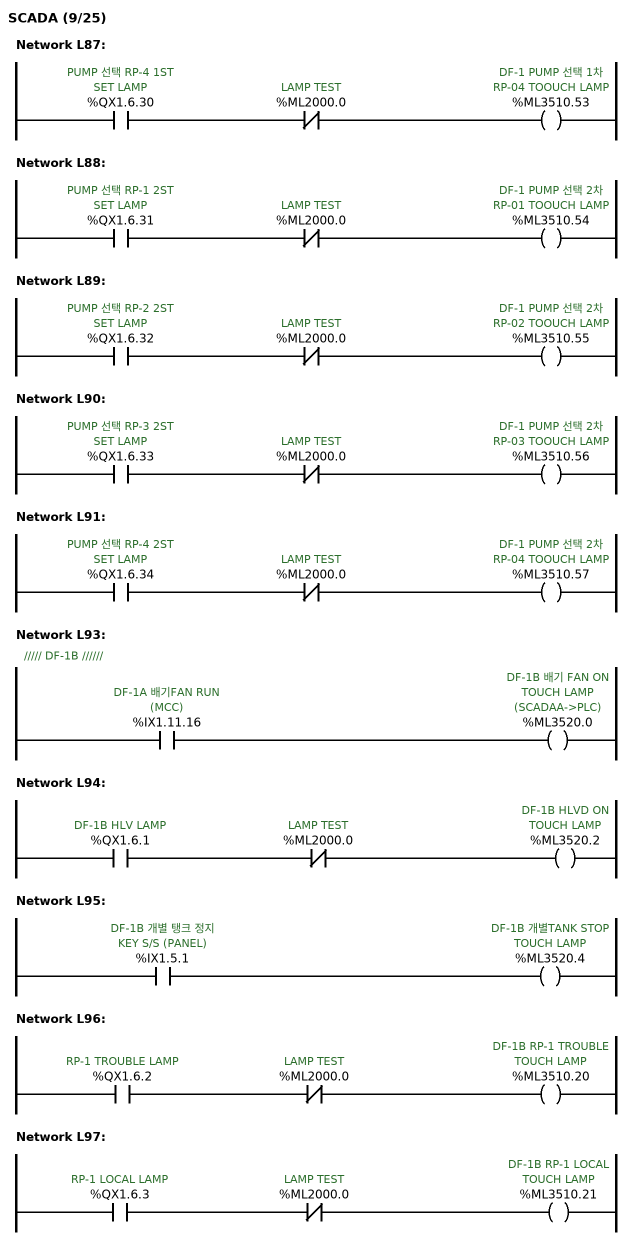
(* [picture p48: SCADA rungs L87-L97] *)
(* Rung L87 *)
%ML3510.53 := %QX1.6.30 AND NOT %ML2000.0;
(* Rung L88 *)
%ML3510.54 := %QX1.6.31 AND NOT %ML2000.0;
(* Rung L89 *)
%ML3510.55 := %QX1.6.32 AND NOT %ML2000.0;
(* Rung L90 *)
%ML3510.56 := %QX1.6.33 AND NOT %ML2000.0;
(* Rung L91 *)
%ML3510.57 := %QX1.6.34 AND NOT %ML2000.0;
(* ///// DF-1B ////// *)
(* Rung L93 *)
%ML3520.0 := %IX1.11.16;
(* Rung L94 *)
%ML3520.2 := %QX1.6.1 AND NOT %ML2000.0;
(* Rung L95 *)
%ML3520.4 := %IX1.5.1;
(* Rung L96 *)
%ML3510.20 := %QX1.6.2 AND NOT %ML2000.0;
(* Rung L97 *)
%ML3510.21 := %QX1.6.3 AND NOT %ML2000.0;

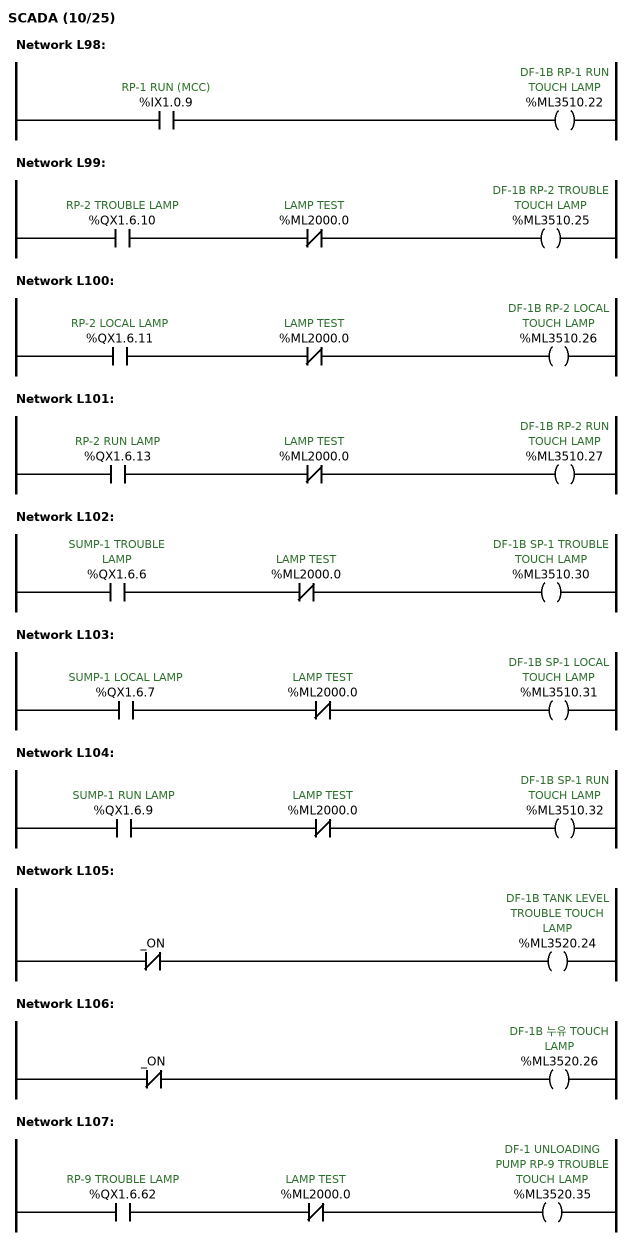
(* Rung L98 *)
%ML3510.22 := %IX1.0.9;
(* Rung L99 *)
%ML3510.25 := %QX1.6.10 AND NOT %ML2000.0;
(* Rung L100 *)
%ML3510.26 := %QX1.6.11 AND NOT %ML2000.0;
(* Rung L101 *)
%ML3510.27 := %QX1.6.13 AND NOT %ML2000.0;
(* Rung L102 *)
%ML3510.30 := %QX1.6.6 AND NOT %ML2000.0;
(* Rung L103 *)
%ML3510.31 := %QX1.6.7 AND NOT %ML2000.0;
(* Rung L104 *)
%ML3510.32 := %QX1.6.9 AND NOT %ML2000.0;
(* Rung L105 *)
%ML3520.24 := NOT _ON;
(* Rung L106 *)
%ML3520.26 := NOT _ON;
(* Rung L107 *)
%ML3520.35 := %QX1.6.62 AND NOT %ML2000.0;

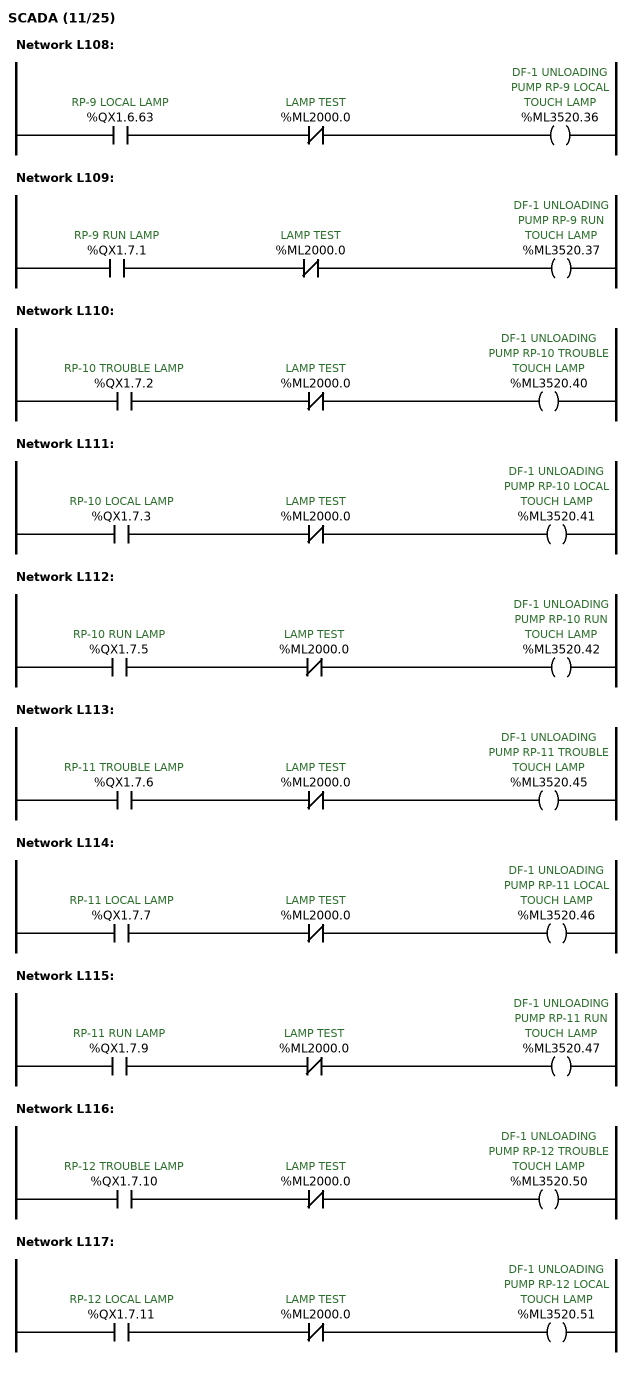
(* Rung L108 *)
%ML3520.36 := %QX1.6.63 AND NOT %ML2000.0;
(* Rung L109 *)
%ML3520.37 := %QX1.7.1 AND NOT %ML2000.0;
(* Rung L110 *)
%ML3520.40 := %QX1.7.2 AND NOT %ML2000.0;
(* Rung L111 *)
%ML3520.41 := %QX1.7.3 AND NOT %ML2000.0;
(* Rung L112 *)
%ML3520.42 := %QX1.7.5 AND NOT %ML2000.0;
(* Rung L113 *)
%ML3520.45 := %QX1.7.6 AND NOT %ML2000.0;
(* Rung L114 *)
%ML3520.46 := %QX1.7.7 AND NOT %ML2000.0;
(* Rung L115 *)
%ML3520.47 := %QX1.7.9 AND NOT %ML2000.0;
(* Rung L116 *)
%ML3520.50 := %QX1.7.10 AND NOT %ML2000.0;
(* Rung L117 *)
%ML3520.51 := %QX1.7.11 AND NOT %ML2000.0;

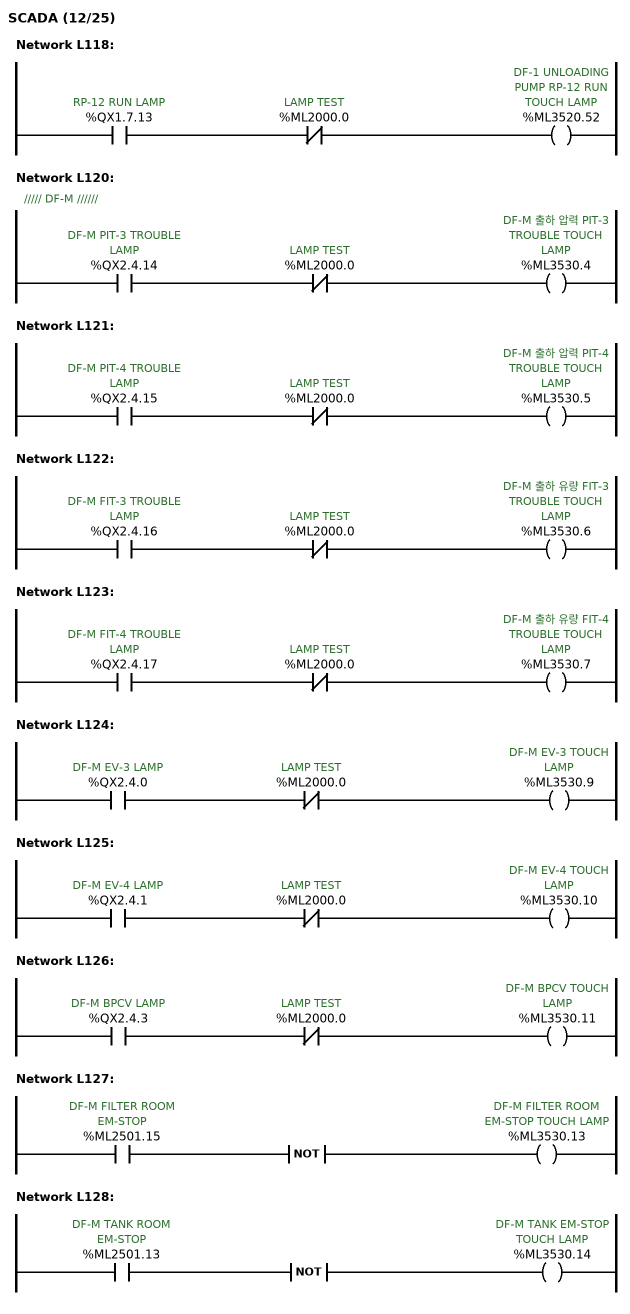
(* Rung L118 *)
%ML3520.52 := %QX1.7.13 AND NOT %ML2000.0;
(* ///// DF-M ////// *)
(* Rung L120 *)
%ML3530.4 := %QX2.4.14 AND NOT %ML2000.0;
(* Rung L121 *)
%ML3530.5 := %QX2.4.15 AND NOT %ML2000.0;
(* Rung L122 *)
%ML3530.6 := %QX2.4.16 AND NOT %ML2000.0;
(* Rung L123 *)
%ML3530.7 := %QX2.4.17 AND NOT %ML2000.0;
(* Rung L124 *)
%ML3530.9 := %QX2.4.0 AND NOT %ML2000.0;
(* Rung L125 *)
%ML3530.10 := %QX2.4.1 AND NOT %ML2000.0;
(* Rung L126 *)
%ML3530.11 := %QX2.4.3 AND NOT %ML2000.0;
(* Rung L127 *)
%ML3530.13 := NOT %ML2501.15;
(* Rung L128 *)
%ML3530.14 := NOT %ML2501.13;

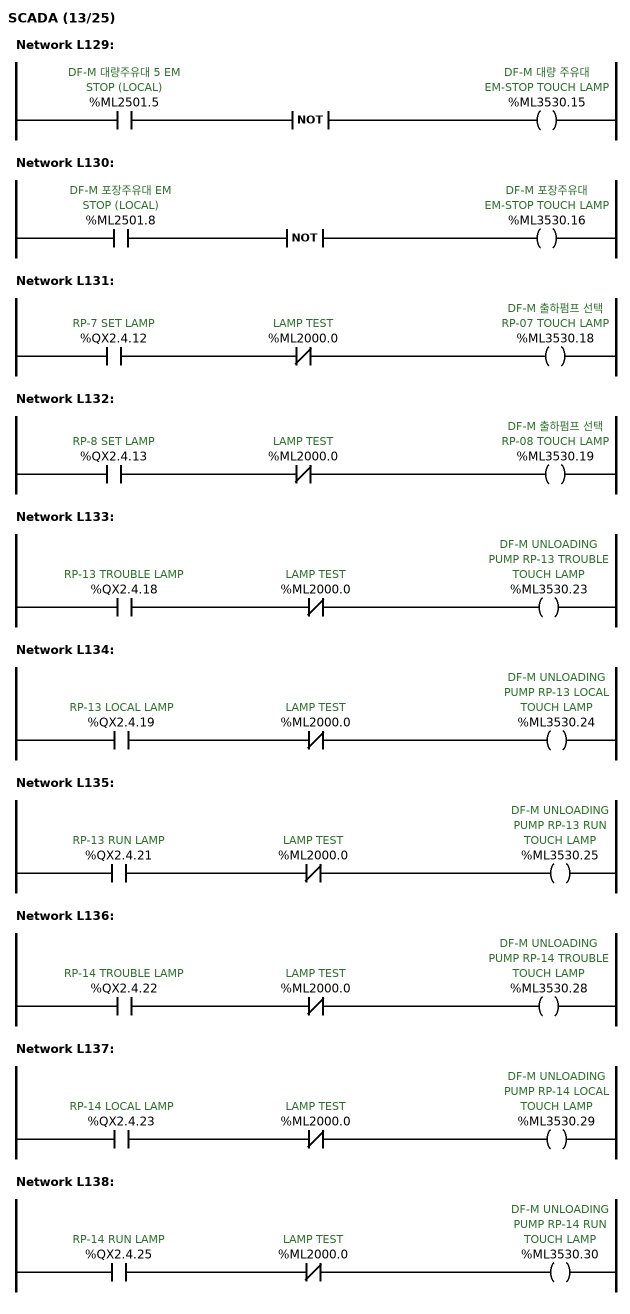
(* Rung L129 *)
%ML3530.15 := NOT %ML2501.5;
(* Rung L130 *)
%ML3530.16 := NOT %ML2501.8;
(* Rung L131 *)
%ML3530.18 := %QX2.4.12 AND NOT %ML2000.0;
(* Rung L132 *)
%ML3530.19 := %QX2.4.13 AND NOT %ML2000.0;
(* Rung L133 *)
%ML3530.23 := %QX2.4.18 AND NOT %ML2000.0;
(* Rung L134 *)
%ML3530.24 := %QX2.4.19 AND NOT %ML2000.0;
(* Rung L135 *)
%ML3530.25 := %QX2.4.21 AND NOT %ML2000.0;
(* Rung L136 *)
%ML3530.28 := %QX2.4.22 AND NOT %ML2000.0;
(* Rung L137 *)
%ML3530.29 := %QX2.4.23 AND NOT %ML2000.0;
(* Rung L138 *)
%ML3530.30 := %QX2.4.25 AND NOT %ML2000.0;

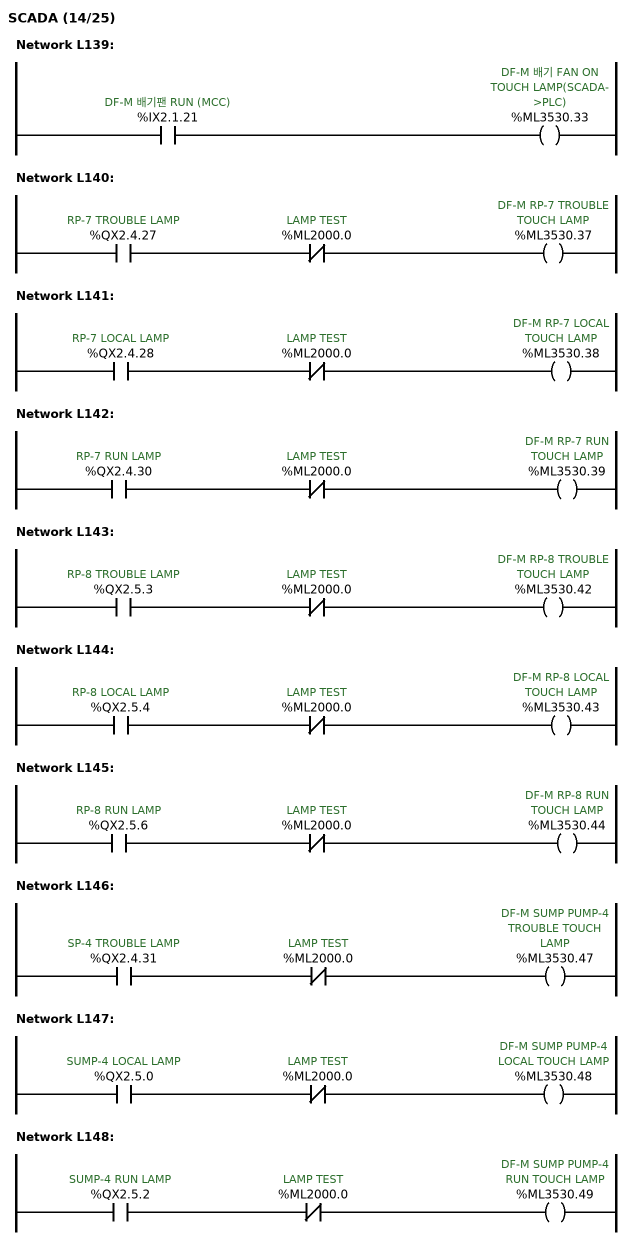
(* Rung L139 *)
%ML3530.33 := %IX2.1.21;
(* Rung L140 *)
%ML3530.37 := %QX2.4.27 AND NOT %ML2000.0;
(* Rung L141 *)
%ML3530.38 := %QX2.4.28 AND NOT %ML2000.0;
(* Rung L142 *)
%ML3530.39 := %QX2.4.30 AND NOT %ML2000.0;
(* Rung L143 *)
%ML3530.42 := %QX2.5.3 AND NOT %ML2000.0;
(* Rung L144 *)
%ML3530.43 := %QX2.5.4 AND NOT %ML2000.0;
(* Rung L145 *)
%ML3530.44 := %QX2.5.6 AND NOT %ML2000.0;
(* Rung L146 *)
%ML3530.47 := %QX2.4.31 AND NOT %ML2000.0;
(* Rung L147 *)
%ML3530.48 := %QX2.5.0 AND NOT %ML2000.0;
(* Rung L148 *)
%ML3530.49 := %QX2.5.2 AND NOT %ML2000.0;

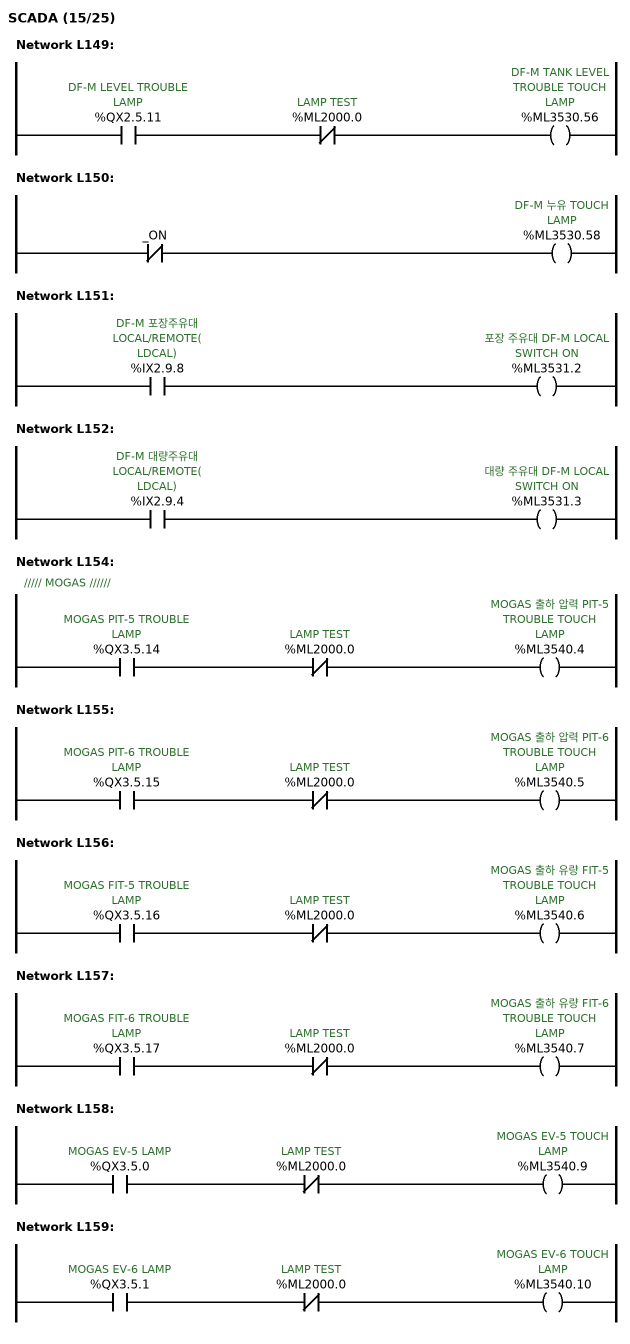
(* Rung L149 *)
%ML3530.56 := %QX2.5.11 AND NOT %ML2000.0;
(* Rung L150 *)
%ML3530.58 := NOT _ON;
(* Rung L151 *)
%ML3531.2 := %IX2.9.8;
(* Rung L152 *)
%ML3531.3 := %IX2.9.4;
(* ///// MOGAS ////// *)
(* Rung L154 *)
%ML3540.4 := %QX3.5.14 AND NOT %ML2000.0;
(* Rung L155 *)
%ML3540.5 := %QX3.5.15 AND NOT %ML2000.0;
(* Rung L156 *)
%ML3540.6 := %QX3.5.16 AND NOT %ML2000.0;
(* Rung L157 *)
%ML3540.7 := %QX3.5.17 AND NOT %ML2000.0;
(* Rung L158 *)
%ML3540.9 := %QX3.5.0 AND NOT %ML2000.0;
(* Rung L159 *)
%ML3540.10 := %QX3.5.1 AND NOT %ML2000.0;

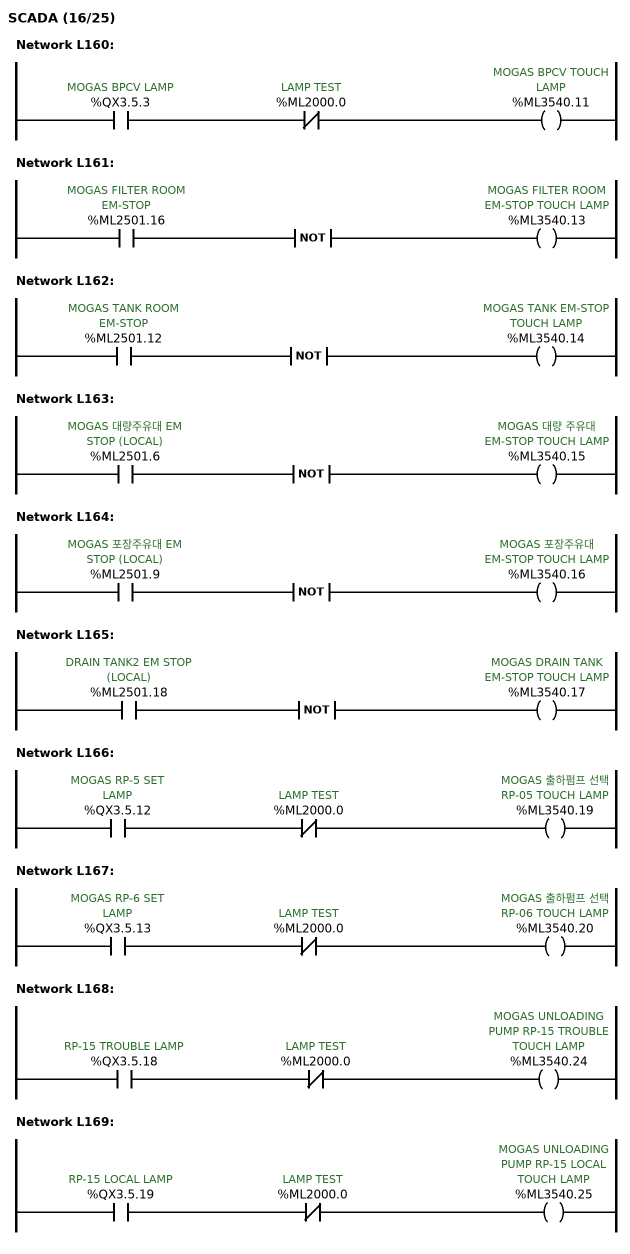
(* Rung L160 *)
%ML3540.11 := %QX3.5.3 AND NOT %ML2000.0;
(* Rung L161 *)
%ML3540.13 := NOT %ML2501.16;
(* Rung L162 *)
%ML3540.14 := NOT %ML2501.12;
(* Rung L163 *)
%ML3540.15 := NOT %ML2501.6;
(* Rung L164 *)
%ML3540.16 := NOT %ML2501.9;
(* Rung L165 *)
%ML3540.17 := NOT %ML2501.18;
(* Rung L166 *)
%ML3540.19 := %QX3.5.12 AND NOT %ML2000.0;
(* Rung L167 *)
%ML3540.20 := %QX3.5.13 AND NOT %ML2000.0;
(* Rung L168 *)
%ML3540.24 := %QX3.5.18 AND NOT %ML2000.0;
(* Rung L169 *)
%ML3540.25 := %QX3.5.19 AND NOT %ML2000.0;

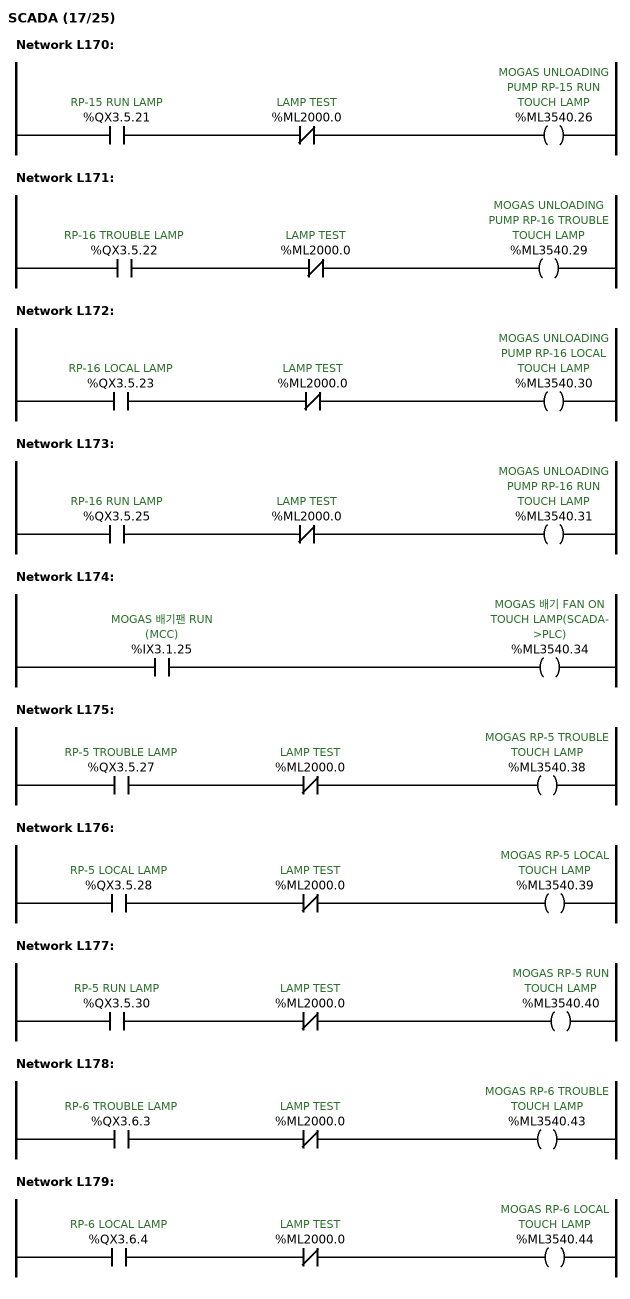
(* Rung L170 *)
%ML3540.26 := %QX3.5.21 AND NOT %ML2000.0;
(* Rung L171 *)
%ML3540.29 := %QX3.5.22 AND NOT %ML2000.0;
(* Rung L172 *)
%ML3540.30 := %QX3.5.23 AND NOT %ML2000.0;
(* Rung L173 *)
%ML3540.31 := %QX3.5.25 AND NOT %ML2000.0;
(* Rung L174 *)
%ML3540.34 := %IX3.1.25;
(* Rung L175 *)
%ML3540.38 := %QX3.5.27 AND NOT %ML2000.0;
(* Rung L176 *)
%ML3540.39 := %QX3.5.28 AND NOT %ML2000.0;
(* Rung L177 *)
%ML3540.40 := %QX3.5.30 AND NOT %ML2000.0;
(* Rung L178 *)
%ML3540.43 := %QX3.6.3 AND NOT %ML2000.0;
(* Rung L179 *)
%ML3540.44 := %QX3.6.4 AND NOT %ML2000.0;

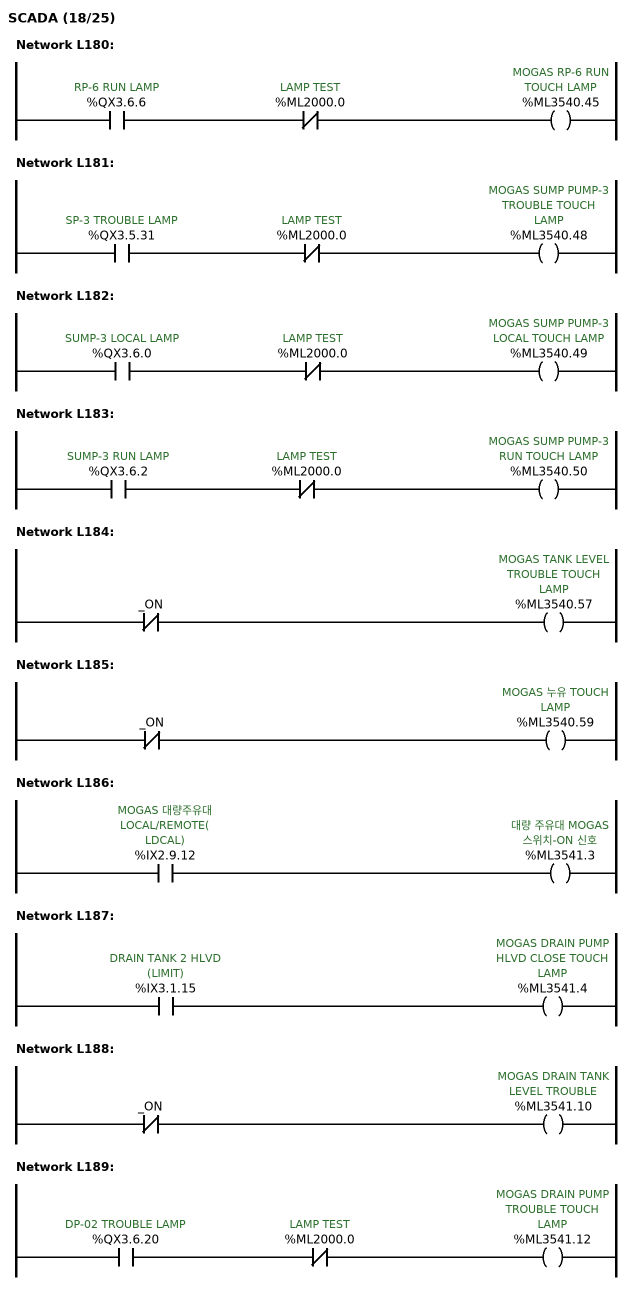
(* Rung L180 *)
%ML3540.45 := %QX3.6.6 AND NOT %ML2000.0;
(* Rung L181 *)
%ML3540.48 := %QX3.5.31 AND NOT %ML2000.0;
(* Rung L182 *)
%ML3540.49 := %QX3.6.0 AND NOT %ML2000.0;
(* Rung L183 *)
%ML3540.50 := %QX3.6.2 AND NOT %ML2000.0;
(* Rung L184 *)
%ML3540.57 := NOT _ON;
(* Rung L185 *)
%ML3540.59 := NOT _ON;
(* Rung L186 *)
%ML3541.3 := %IX2.9.12;
(* Rung L187 *)
%ML3541.4 := %IX3.1.15;
(* Rung L188 *)
%ML3541.10 := NOT _ON;
(* Rung L189 *)
%ML3541.12 := %QX3.6.20 AND NOT %ML2000.0;

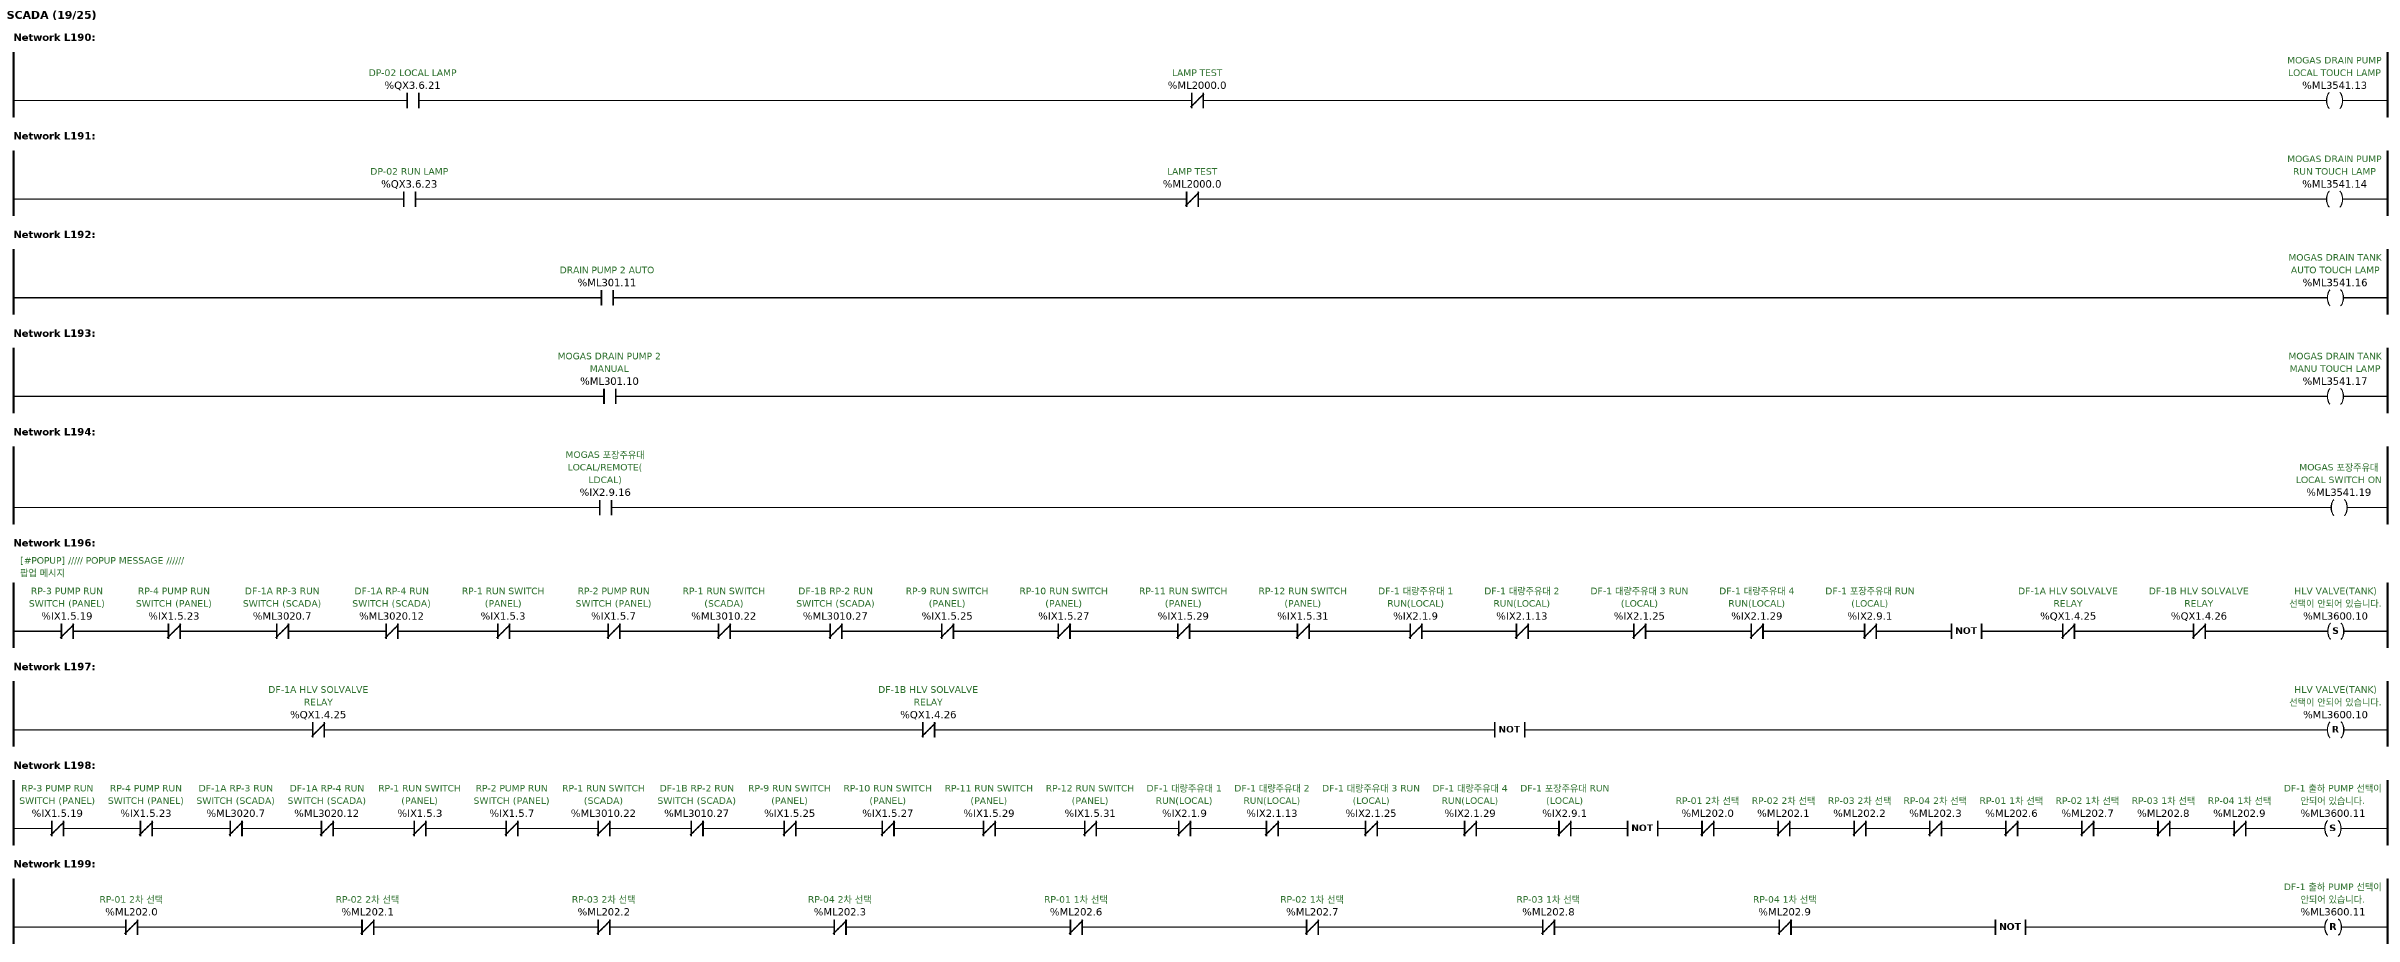
(* Rung L190 *)
%ML3541.13 := %QX3.6.21 AND NOT %ML2000.0;
(* Rung L191 *)
%ML3541.14 := %QX3.6.23 AND NOT %ML2000.0;
(* Rung L192 *)
%ML3541.16 := %ML301.11;
(* Rung L193 *)
%ML3541.17 := %ML301.10;
(* Rung L194 *)
%ML3541.19 := %IX2.9.16;
(* [#POPUP] ///// POPUP MESSAGE ////// *)
(* Rung L196 *)
IF NOT (NOT %IX1.5.19 AND NOT %IX1.5.23 AND NOT %ML3020.7 AND NOT %ML3020.12 AND NOT %IX1.5.3 AND NOT %IX1.5.7 AND NOT %ML3010.22 AND NOT %ML3010.27 AND NOT %IX1.5.25 AND NOT %IX1.5.27 AND NOT %IX1.5.29 AND NOT %IX1.5.31 AND NOT %IX2.1.9 AND NOT %IX2.1.13 AND NOT %IX2.1.25 AND NOT %IX2.1.29 AND NOT %IX2.9.1) AND NOT %QX1.4.25 AND NOT %QX1.4.26 THEN
    %ML3600.10 := TRUE;
END_IF;
(* 팝업 메시지 *)
(* Rung L197 *)
IF NOT (NOT %QX1.4.25 AND NOT %QX1.4.26) THEN %ML3600.10 := FALSE; END_IF;
(* Rung L198 *)
IF NOT (NOT %IX1.5.19 AND NOT %IX1.5.23 AND NOT %ML3020.7 AND NOT %ML3020.12 AND NOT %IX1.5.3 AND NOT %IX1.5.7 AND NOT %ML3010.22 AND NOT %ML3010.27 AND NOT %IX1.5.25 AND NOT %IX1.5.27 AND NOT %IX1.5.29 AND NOT %IX1.5.31 AND NOT %IX2.1.9 AND NOT %IX2.1.13 AND NOT %IX2.1.25 AND NOT %IX2.1.29 AND NOT %IX2.9.1) AND NOT %ML202.0 AND NOT %ML202.1 AND NOT %ML202.2 AND NOT %ML202.3 AND NOT %ML202.6 AND NOT %ML202.7 AND NOT %ML202.8 AND NOT %ML202.9 THEN
    %ML3600.11 := TRUE;
END_IF;
(* Rung L199 *)
IF NOT (NOT %ML202.0 AND NOT %ML202.1 AND NOT %ML202.2 AND NOT %ML202.3 AND NOT %ML202.6 AND NOT %ML202.7 AND NOT %ML202.8 AND NOT %ML202.9) THEN
    %ML3600.11 := FALSE;
END_IF;

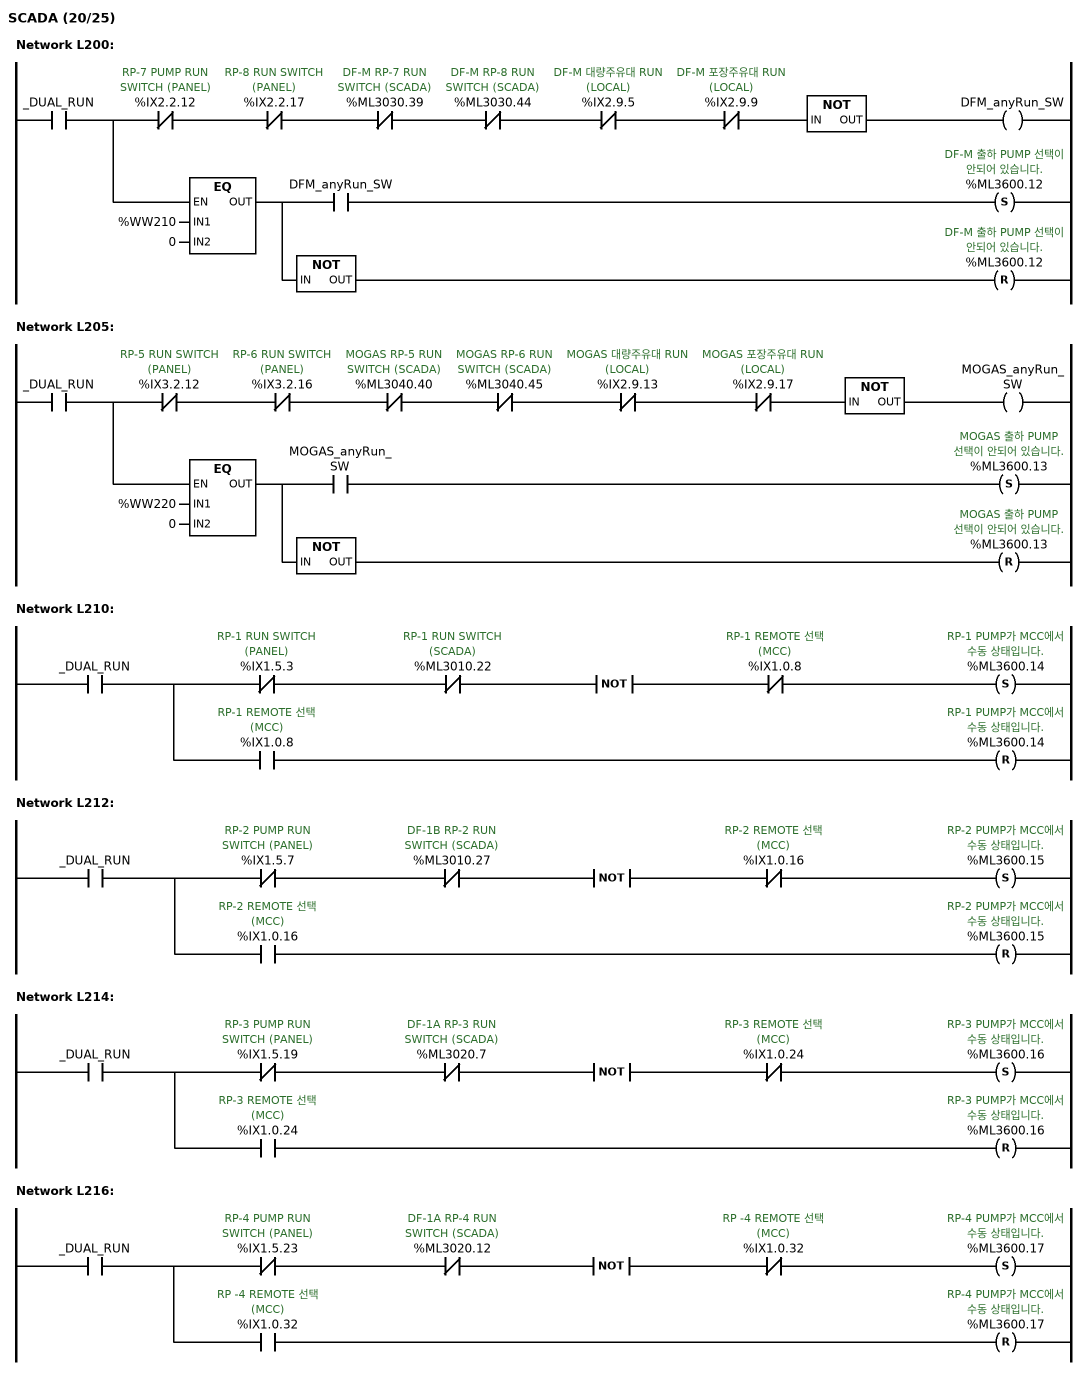
(* Rung L200 *)
DFM_anyRun_SW := NOT (_DUAL_RUN AND NOT %IX2.2.12 AND NOT %IX2.2.17 AND NOT %ML3030.39 AND NOT %ML3030.44 AND NOT %IX2.9.5 AND NOT %IX2.9.9);
IF _DUAL_RUN THEN _t1 := %WW210 = 0; END_IF;
IF _t1 AND DFM_anyRun_SW THEN %ML3600.12 := TRUE; END_IF;
IF NOT _t1 THEN %ML3600.12 := FALSE; END_IF;
(* Rung L205 *)
MOGAS_anyRun_SW := NOT (_DUAL_RUN AND NOT %IX3.2.12 AND NOT %IX3.2.16 AND NOT %ML3040.40 AND NOT %ML3040.45 AND NOT %IX2.9.13 AND NOT %IX2.9.17);
IF _DUAL_RUN THEN _t2 := %WW220 = 0; END_IF;
IF _t2 AND MOGAS_anyRun_SW THEN %ML3600.13 := TRUE; END_IF;
IF NOT _t2 THEN %ML3600.13 := FALSE; END_IF;
(* Rung L210 *)
IF NOT (_DUAL_RUN AND NOT %IX1.5.3 AND NOT %ML3010.22) AND NOT %IX1.0.8 THEN %ML3600.14 := TRUE; END_IF;
IF _DUAL_RUN AND %IX1.0.8 THEN %ML3600.14 := FALSE; END_IF;
(* Rung L212 *)
IF NOT (_DUAL_RUN AND NOT %IX1.5.7 AND NOT %ML3010.27) AND NOT %IX1.0.16 THEN %ML3600.15 := TRUE; END_IF;
IF _DUAL_RUN AND %IX1.0.16 THEN %ML3600.15 := FALSE; END_IF;
(* Rung L214 *)
IF NOT (_DUAL_RUN AND NOT %IX1.5.19 AND NOT %ML3020.7) AND NOT %IX1.0.24 THEN %ML3600.16 := TRUE; END_IF;
IF _DUAL_RUN AND %IX1.0.24 THEN %ML3600.16 := FALSE; END_IF;
(* Rung L216 *)
IF NOT (_DUAL_RUN AND NOT %IX1.5.23 AND NOT %ML3020.12) AND NOT %IX1.0.32 THEN %ML3600.17 := TRUE; END_IF;
IF _DUAL_RUN AND %IX1.0.32 THEN %ML3600.17 := FALSE; END_IF;

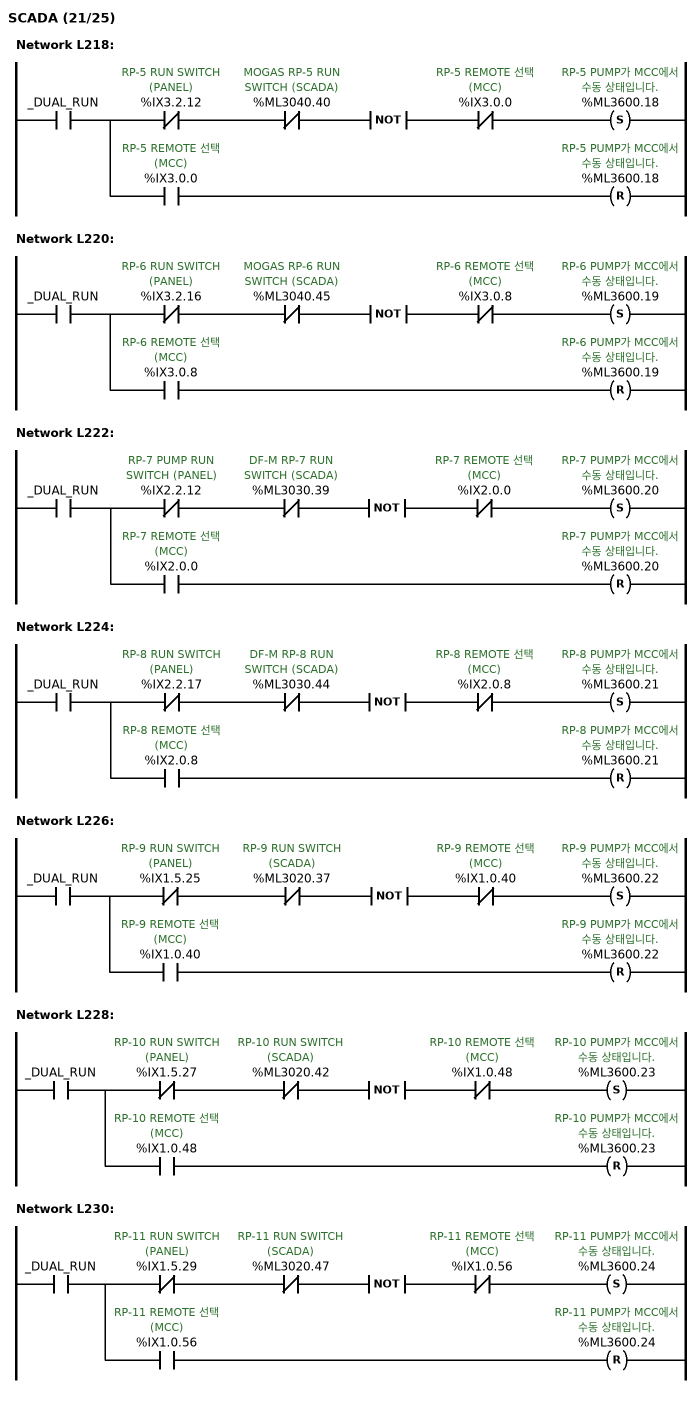
(* Rung L218 *)
IF NOT (_DUAL_RUN AND NOT %IX3.2.12 AND NOT %ML3040.40) AND NOT %IX3.0.0 THEN %ML3600.18 := TRUE; END_IF;
IF _DUAL_RUN AND %IX3.0.0 THEN %ML3600.18 := FALSE; END_IF;
(* Rung L220 *)
IF NOT (_DUAL_RUN AND NOT %IX3.2.16 AND NOT %ML3040.45) AND NOT %IX3.0.8 THEN %ML3600.19 := TRUE; END_IF;
IF _DUAL_RUN AND %IX3.0.8 THEN %ML3600.19 := FALSE; END_IF;
(* Rung L222 *)
IF NOT (_DUAL_RUN AND NOT %IX2.2.12 AND NOT %ML3030.39) AND NOT %IX2.0.0 THEN %ML3600.20 := TRUE; END_IF;
IF _DUAL_RUN AND %IX2.0.0 THEN %ML3600.20 := FALSE; END_IF;
(* Rung L224 *)
IF NOT (_DUAL_RUN AND NOT %IX2.2.17 AND NOT %ML3030.44) AND NOT %IX2.0.8 THEN %ML3600.21 := TRUE; END_IF;
IF _DUAL_RUN AND %IX2.0.8 THEN %ML3600.21 := FALSE; END_IF;
(* Rung L226 *)
IF NOT (_DUAL_RUN AND NOT %IX1.5.25 AND NOT %ML3020.37) AND NOT %IX1.0.40 THEN %ML3600.22 := TRUE; END_IF;
IF _DUAL_RUN AND %IX1.0.40 THEN %ML3600.22 := FALSE; END_IF;
(* Rung L228 *)
IF NOT (_DUAL_RUN AND NOT %IX1.5.27 AND NOT %ML3020.42) AND NOT %IX1.0.48 THEN %ML3600.23 := TRUE; END_IF;
IF _DUAL_RUN AND %IX1.0.48 THEN %ML3600.23 := FALSE; END_IF;
(* Rung L230 *)
IF NOT (_DUAL_RUN AND NOT %IX1.5.29 AND NOT %ML3020.47) AND NOT %IX1.0.56 THEN %ML3600.24 := TRUE; END_IF;
IF _DUAL_RUN AND %IX1.0.56 THEN %ML3600.24 := FALSE; END_IF;

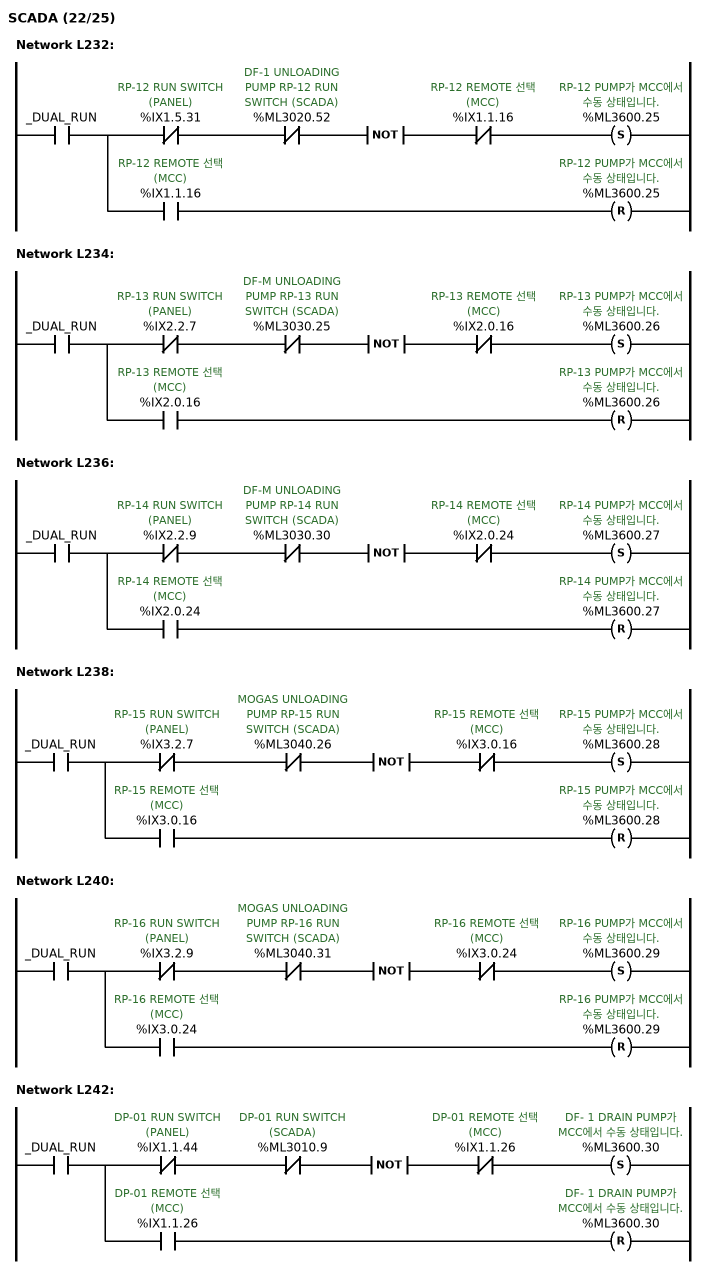
(* Rung L232 *)
IF NOT (_DUAL_RUN AND NOT %IX1.5.31 AND NOT %ML3020.52) AND NOT %IX1.1.16 THEN %ML3600.25 := TRUE; END_IF;
IF _DUAL_RUN AND %IX1.1.16 THEN %ML3600.25 := FALSE; END_IF;
(* Rung L234 *)
IF NOT (_DUAL_RUN AND NOT %IX2.2.7 AND NOT %ML3030.25) AND NOT %IX2.0.16 THEN %ML3600.26 := TRUE; END_IF;
IF _DUAL_RUN AND %IX2.0.16 THEN %ML3600.26 := FALSE; END_IF;
(* Rung L236 *)
IF NOT (_DUAL_RUN AND NOT %IX2.2.9 AND NOT %ML3030.30) AND NOT %IX2.0.24 THEN %ML3600.27 := TRUE; END_IF;
IF _DUAL_RUN AND %IX2.0.24 THEN %ML3600.27 := FALSE; END_IF;
(* Rung L238 *)
IF NOT (_DUAL_RUN AND NOT %IX3.2.7 AND NOT %ML3040.26) AND NOT %IX3.0.16 THEN %ML3600.28 := TRUE; END_IF;
IF _DUAL_RUN AND %IX3.0.16 THEN %ML3600.28 := FALSE; END_IF;
(* Rung L240 *)
IF NOT (_DUAL_RUN AND NOT %IX3.2.9 AND NOT %ML3040.31) AND NOT %IX3.0.24 THEN %ML3600.29 := TRUE; END_IF;
IF _DUAL_RUN AND %IX3.0.24 THEN %ML3600.29 := FALSE; END_IF;
(* Rung L242 *)
IF NOT (_DUAL_RUN AND NOT %IX1.1.44 AND NOT %ML3010.9) AND NOT %IX1.1.26 THEN %ML3600.30 := TRUE; END_IF;
IF _DUAL_RUN AND %IX1.1.26 THEN %ML3600.30 := FALSE; END_IF;

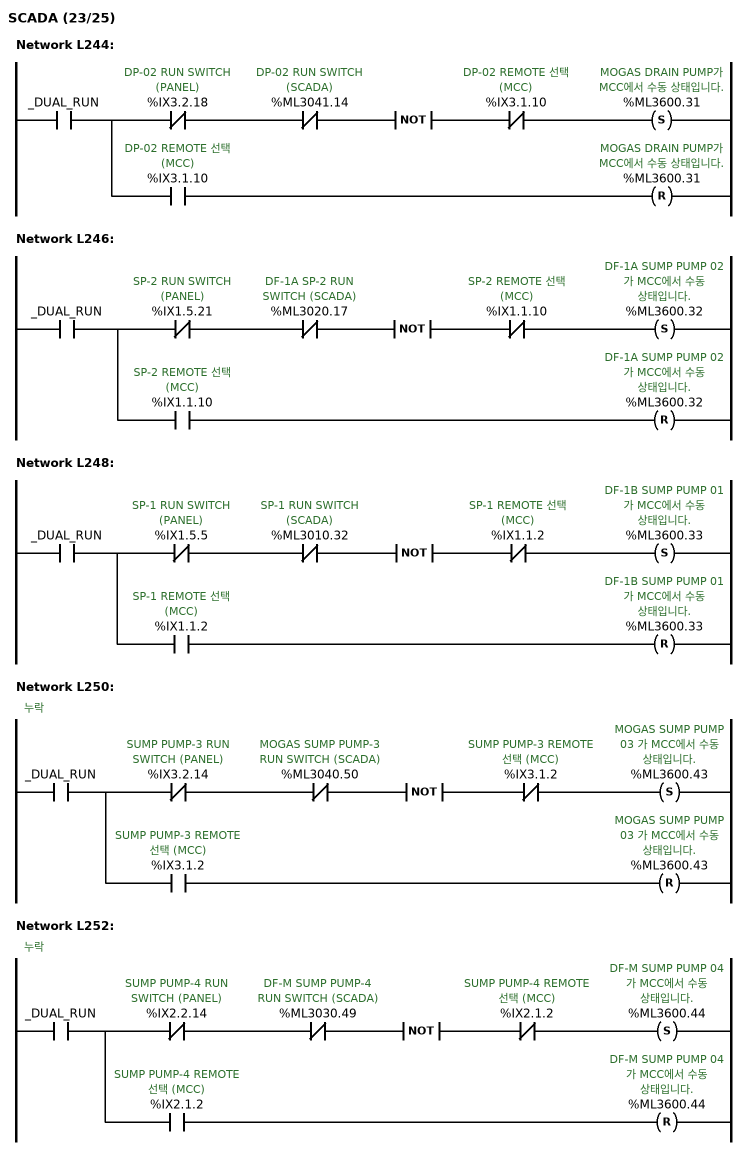
(* Rung L244 *)
IF NOT (_DUAL_RUN AND NOT %IX3.2.18 AND NOT %ML3041.14) AND NOT %IX3.1.10 THEN %ML3600.31 := TRUE; END_IF;
IF _DUAL_RUN AND %IX3.1.10 THEN %ML3600.31 := FALSE; END_IF;
(* Rung L246 *)
IF NOT (_DUAL_RUN AND NOT %IX1.5.21 AND NOT %ML3020.17) AND NOT %IX1.1.10 THEN %ML3600.32 := TRUE; END_IF;
IF _DUAL_RUN AND %IX1.1.10 THEN %ML3600.32 := FALSE; END_IF;
(* Rung L248 *)
IF NOT (_DUAL_RUN AND NOT %IX1.5.5 AND NOT %ML3010.32) AND NOT %IX1.1.2 THEN %ML3600.33 := TRUE; END_IF;
IF _DUAL_RUN AND %IX1.1.2 THEN %ML3600.33 := FALSE; END_IF;
(* Rung L250 *)
IF NOT (_DUAL_RUN AND NOT %IX3.2.14 AND NOT %ML3040.50) AND NOT %IX3.1.2 THEN %ML3600.43 := TRUE; END_IF;
IF _DUAL_RUN AND %IX3.1.2 THEN %ML3600.43 := FALSE; END_IF;
(* 누락 *)
(* Rung L252 *)
IF NOT (_DUAL_RUN AND NOT %IX2.2.14 AND NOT %ML3030.49) AND NOT %IX2.1.2 THEN %ML3600.44 := TRUE; END_IF;
IF _DUAL_RUN AND %IX2.1.2 THEN %ML3600.44 := FALSE; END_IF;
(* 누락 *)

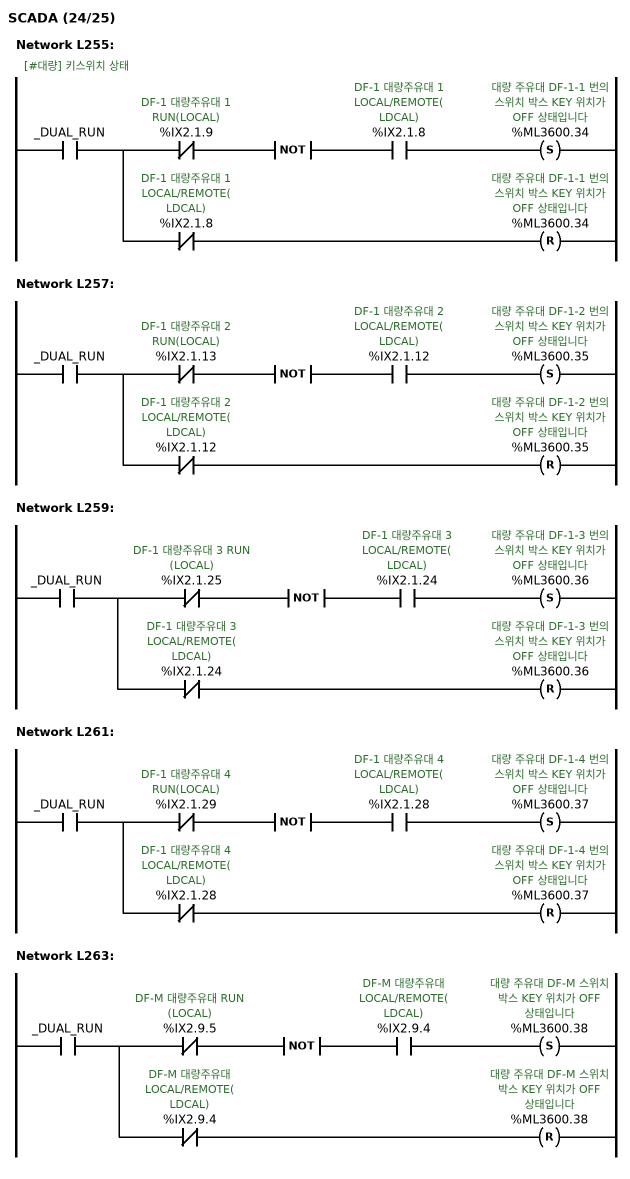
(* [#대량] 키스위치 상태 *)
(* Rung L255 *)
IF NOT (_DUAL_RUN AND NOT %IX2.1.9) AND %IX2.1.8 THEN %ML3600.34 := TRUE; END_IF;
IF _DUAL_RUN AND NOT %IX2.1.8 THEN %ML3600.34 := FALSE; END_IF;
(* Rung L257 *)
IF NOT (_DUAL_RUN AND NOT %IX2.1.13) AND %IX2.1.12 THEN %ML3600.35 := TRUE; END_IF;
IF _DUAL_RUN AND NOT %IX2.1.12 THEN %ML3600.35 := FALSE; END_IF;
(* Rung L259 *)
IF NOT (_DUAL_RUN AND NOT %IX2.1.25) AND %IX2.1.24 THEN %ML3600.36 := TRUE; END_IF;
IF _DUAL_RUN AND NOT %IX2.1.24 THEN %ML3600.36 := FALSE; END_IF;
(* Rung L261 *)
IF NOT (_DUAL_RUN AND NOT %IX2.1.29) AND %IX2.1.28 THEN %ML3600.37 := TRUE; END_IF;
IF _DUAL_RUN AND NOT %IX2.1.28 THEN %ML3600.37 := FALSE; END_IF;
(* Rung L263 *)
IF NOT (_DUAL_RUN AND NOT %IX2.9.5) AND %IX2.9.4 THEN %ML3600.38 := TRUE; END_IF;
IF _DUAL_RUN AND NOT %IX2.9.4 THEN %ML3600.38 := FALSE; END_IF;

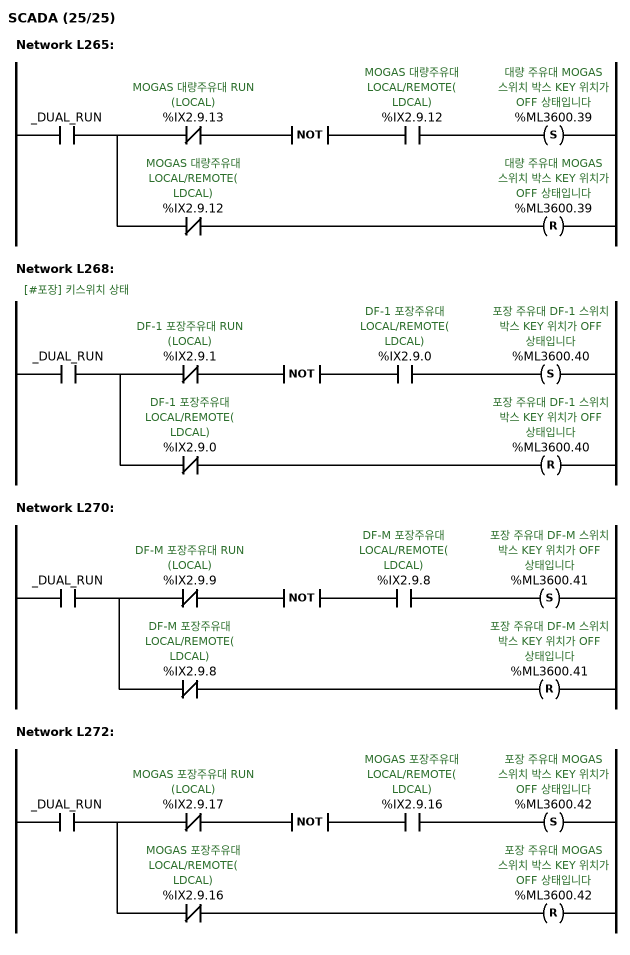
(* Rung L265 *)
IF NOT (_DUAL_RUN AND NOT %IX2.9.13) AND %IX2.9.12 THEN %ML3600.39 := TRUE; END_IF;
IF _DUAL_RUN AND NOT %IX2.9.12 THEN %ML3600.39 := FALSE; END_IF;
(* [#포장] 키스위치 상태 *)
(* Rung L268 *)
IF NOT (_DUAL_RUN AND NOT %IX2.9.1) AND %IX2.9.0 THEN %ML3600.40 := TRUE; END_IF;
IF _DUAL_RUN AND NOT %IX2.9.0 THEN %ML3600.40 := FALSE; END_IF;
(* Rung L270 *)
IF NOT (_DUAL_RUN AND NOT %IX2.9.9) AND %IX2.9.8 THEN %ML3600.41 := TRUE; END_IF;
IF _DUAL_RUN AND NOT %IX2.9.8 THEN %ML3600.41 := FALSE; END_IF;
(* Rung L272 *)
IF NOT (_DUAL_RUN AND NOT %IX2.9.17) AND %IX2.9.16 THEN %ML3600.42 := TRUE; END_IF;
IF _DUAL_RUN AND NOT %IX2.9.16 THEN %ML3600.42 := FALSE; END_IF;
END_PROGRAM

PROGRAM OUT (* task: 스캔 프로그램 *)
VAR
    D10 : BOOL;
    D1000 : BOOL;
    H16 : BOOL;
    INST : FF;
END_VAR
VAR
    _t1 : BOOL;
    _t2 : BOOL;
    _t3 : BOOL;
    _t4 : BOOL;
    _t5 : BOOL;
    _t6 : BOOL;
    _t7 : BOOL;
    _t8 : BOOL;
    _t9 : BOOL;
    _t10 : BOOL;
    _t11 : BOOL;
    _t12 : BOOL;
END_VAR

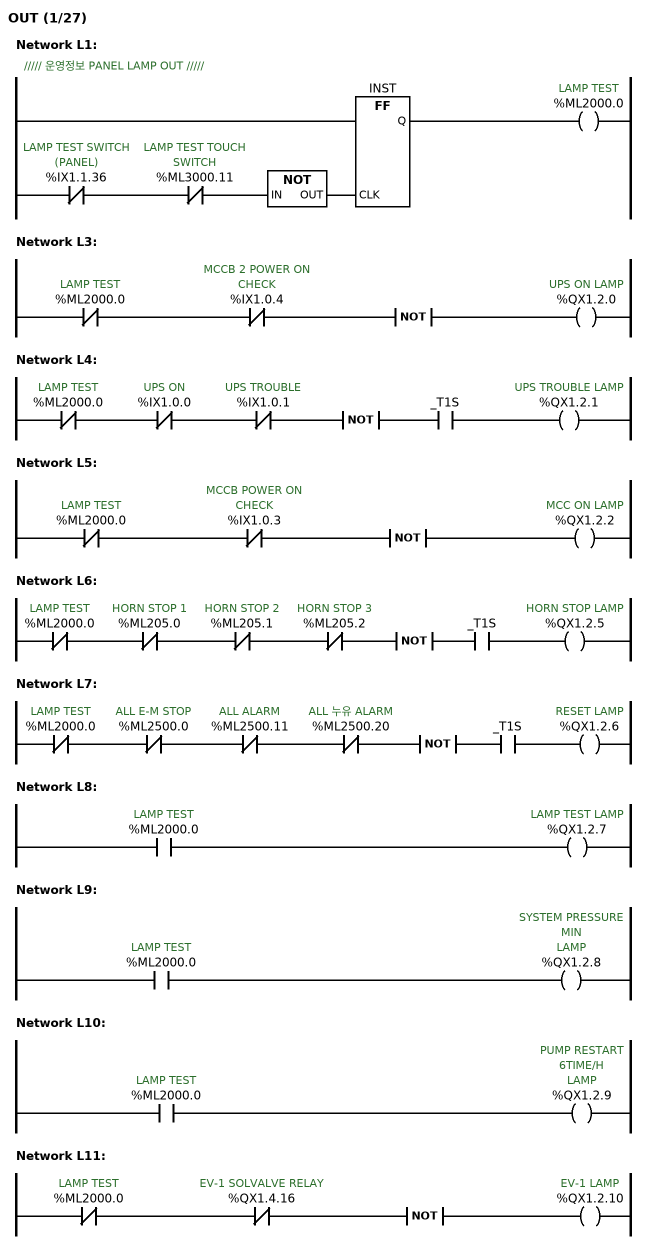
(* ///// 운영정보 PANEL LAMP OUT ///// *)
(* Rung L1 *)
INST(CLK := NOT (NOT %IX1.1.36 AND NOT %ML3000.11));
%ML2000.0 := INST.Q;
(* Rung L3 *)
%QX1.2.0 := NOT (NOT %ML2000.0 AND NOT %IX1.0.4);
(* Rung L4 *)
%QX1.2.1 := NOT (NOT %ML2000.0 AND NOT %IX1.0.0 AND NOT %IX1.0.1) AND _T1S;
(* Rung L5 *)
%QX1.2.2 := NOT (NOT %ML2000.0 AND NOT %IX1.0.3);
(* Rung L6 *)
%QX1.2.5 := NOT (NOT %ML2000.0 AND NOT %ML205.0 AND NOT %ML205.1 AND NOT %ML205.2) AND _T1S;
(* Rung L7 *)
%QX1.2.6 := NOT (NOT %ML2000.0 AND NOT %ML2500.0 AND NOT %ML2500.11 AND NOT %ML2500.20) AND _T1S;
(* Rung L8 *)
%QX1.2.7 := %ML2000.0;
(* Rung L9 *)
%QX1.2.8 := %ML2000.0;
(* Rung L10 *)
%QX1.2.9 := %ML2000.0;
(* Rung L11 *)
%QX1.2.10 := NOT (NOT %ML2000.0 AND NOT %QX1.4.16);

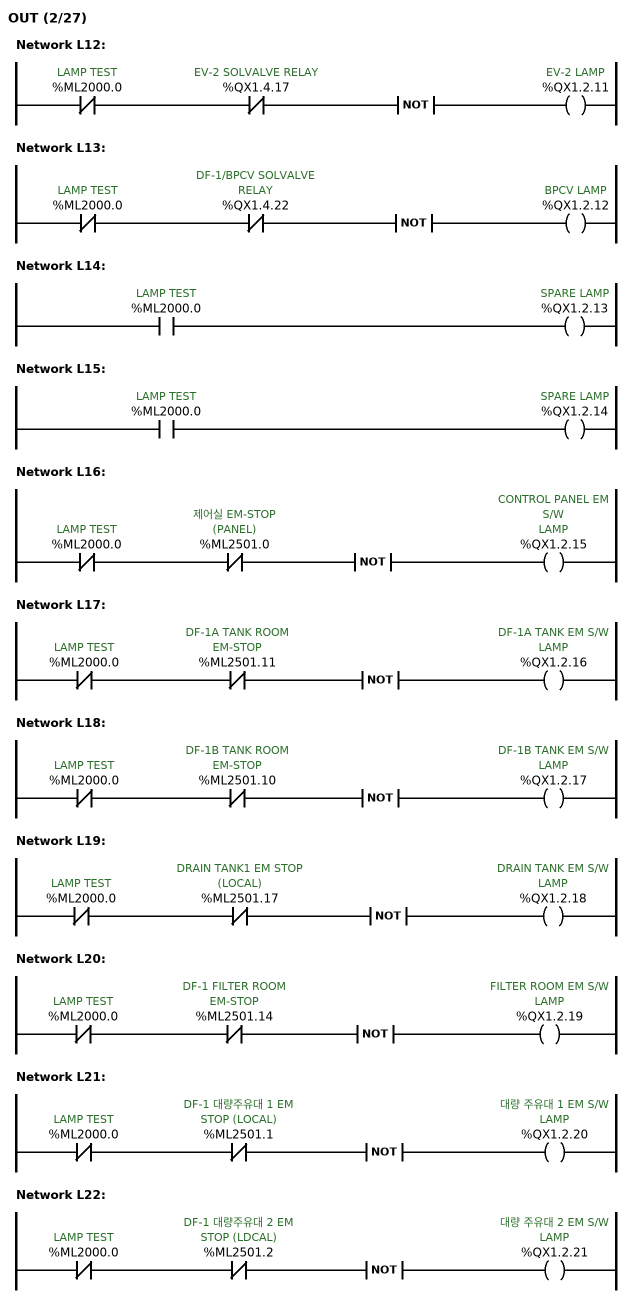
(* Rung L12 *)
%QX1.2.11 := NOT (NOT %ML2000.0 AND NOT %QX1.4.17);
(* Rung L13 *)
%QX1.2.12 := NOT (NOT %ML2000.0 AND NOT %QX1.4.22);
(* Rung L14 *)
%QX1.2.13 := %ML2000.0;
(* Rung L15 *)
%QX1.2.14 := %ML2000.0;
(* Rung L16 *)
%QX1.2.15 := NOT (NOT %ML2000.0 AND NOT %ML2501.0);
(* Rung L17 *)
%QX1.2.16 := NOT (NOT %ML2000.0 AND NOT %ML2501.11);
(* Rung L18 *)
%QX1.2.17 := NOT (NOT %ML2000.0 AND NOT %ML2501.10);
(* Rung L19 *)
%QX1.2.18 := NOT (NOT %ML2000.0 AND NOT %ML2501.17);
(* Rung L20 *)
%QX1.2.19 := NOT (NOT %ML2000.0 AND NOT %ML2501.14);
(* Rung L21 *)
%QX1.2.20 := NOT (NOT %ML2000.0 AND NOT %ML2501.1);
(* Rung L22 *)
%QX1.2.21 := NOT (NOT %ML2000.0 AND NOT %ML2501.2);

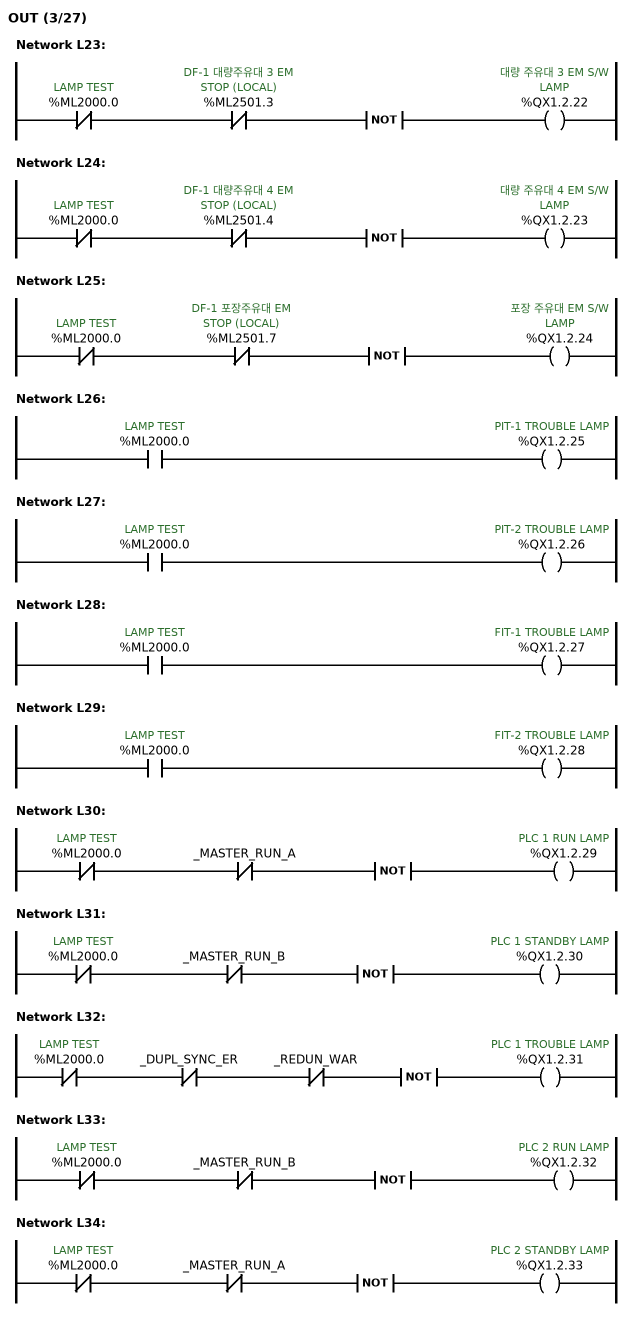
(* Rung L23 *)
%QX1.2.22 := NOT (NOT %ML2000.0 AND NOT %ML2501.3);
(* Rung L24 *)
%QX1.2.23 := NOT (NOT %ML2000.0 AND NOT %ML2501.4);
(* Rung L25 *)
%QX1.2.24 := NOT (NOT %ML2000.0 AND NOT %ML2501.7);
(* Rung L26 *)
%QX1.2.25 := %ML2000.0;
(* Rung L27 *)
%QX1.2.26 := %ML2000.0;
(* Rung L28 *)
%QX1.2.27 := %ML2000.0;
(* Rung L29 *)
%QX1.2.28 := %ML2000.0;
(* Rung L30 *)
%QX1.2.29 := NOT (NOT %ML2000.0 AND NOT _MASTER_RUN_A);
(* Rung L31 *)
%QX1.2.30 := NOT (NOT %ML2000.0 AND NOT _MASTER_RUN_B);
(* Rung L32 *)
%QX1.2.31 := NOT (NOT %ML2000.0 AND NOT _DUPL_SYNC_ER AND NOT _REDUN_WAR);
(* Rung L33 *)
%QX1.2.32 := NOT (NOT %ML2000.0 AND NOT _MASTER_RUN_B);
(* Rung L34 *)
%QX1.2.33 := NOT (NOT %ML2000.0 AND NOT _MASTER_RUN_A);

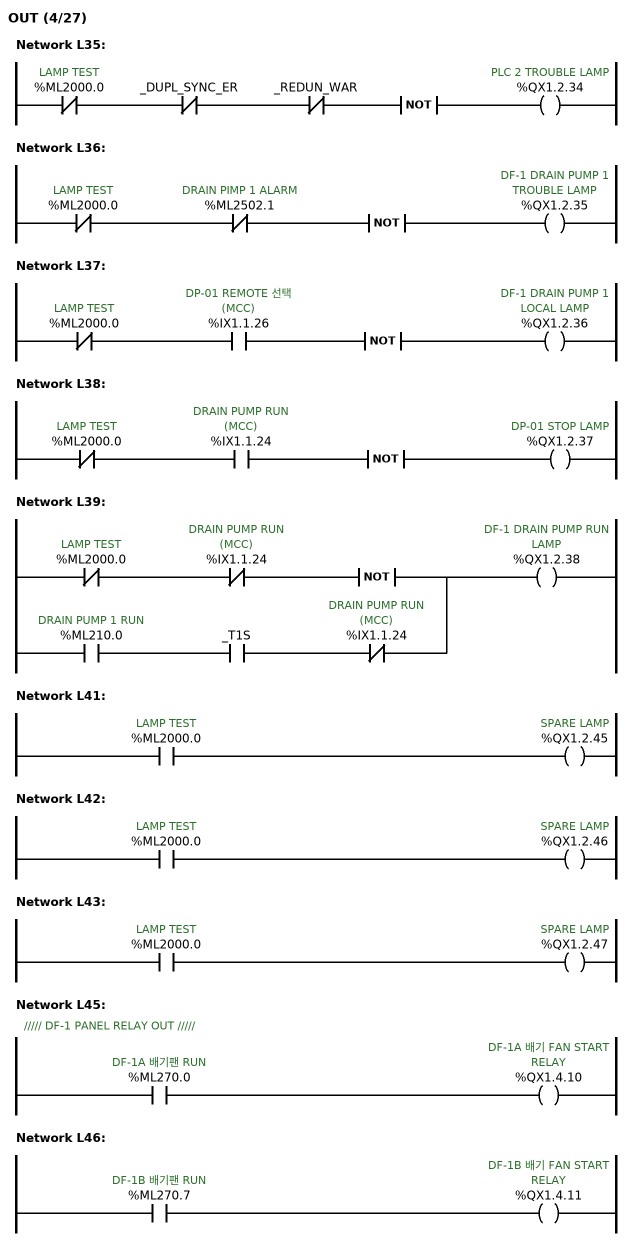
(* Rung L35 *)
%QX1.2.34 := NOT (NOT %ML2000.0 AND NOT _DUPL_SYNC_ER AND NOT _REDUN_WAR);
(* Rung L36 *)
%QX1.2.35 := NOT (NOT %ML2000.0 AND NOT %ML2502.1);
(* Rung L37 *)
%QX1.2.36 := NOT (NOT %ML2000.0 AND %IX1.1.26);
(* Rung L38 *)
%QX1.2.37 := NOT (NOT %ML2000.0 AND %IX1.1.24);
(* Rung L39 *)
%QX1.2.38 := NOT (NOT %ML2000.0 AND NOT %IX1.1.24) OR (%ML210.0 AND _T1S AND NOT %IX1.1.24);
(* Rung L41 *)
%QX1.2.45 := %ML2000.0;
(* Rung L42 *)
%QX1.2.46 := %ML2000.0;
(* Rung L43 *)
%QX1.2.47 := %ML2000.0;
(* ///// DF-1 PANEL RELAY OUT ///// *)
(* Rung L45 *)
%QX1.4.10 := %ML270.0;
(* Rung L46 *)
%QX1.4.11 := %ML270.7;

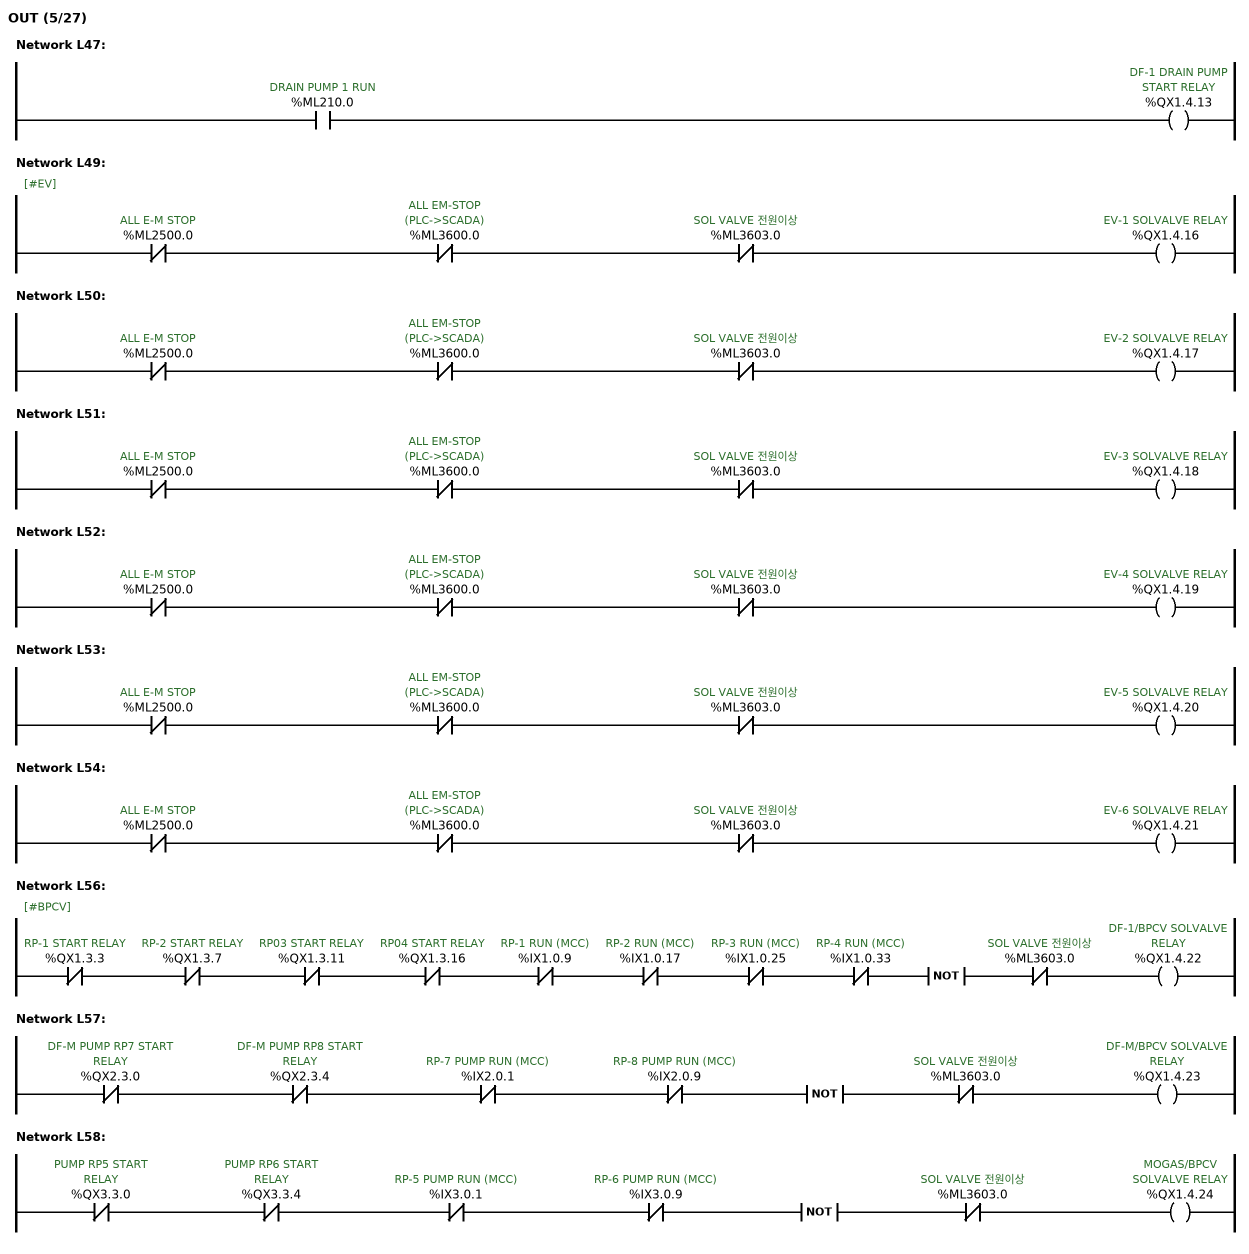
(* Rung L47 *)
%QX1.4.13 := %ML210.0;
(* [#EV] *)
(* Rung L49 *)
%QX1.4.16 := NOT %ML2500.0 AND NOT %ML3600.0 AND NOT %ML3603.0;
(* Rung L50 *)
%QX1.4.17 := NOT %ML2500.0 AND NOT %ML3600.0 AND NOT %ML3603.0;
(* Rung L51 *)
%QX1.4.18 := NOT %ML2500.0 AND NOT %ML3600.0 AND NOT %ML3603.0;
(* Rung L52 *)
%QX1.4.19 := NOT %ML2500.0 AND NOT %ML3600.0 AND NOT %ML3603.0;
(* Rung L53 *)
%QX1.4.20 := NOT %ML2500.0 AND NOT %ML3600.0 AND NOT %ML3603.0;
(* Rung L54 *)
%QX1.4.21 := NOT %ML2500.0 AND NOT %ML3600.0 AND NOT %ML3603.0;
(* [#BPCV] *)
(* Rung L56 *)
%QX1.4.22 := NOT (NOT %QX1.3.3 AND NOT %QX1.3.7 AND NOT %QX1.3.11 AND NOT %QX1.3.16 AND NOT %IX1.0.9 AND NOT %IX1.0.17 AND NOT %IX1.0.25 AND NOT %IX1.0.33) AND NOT %ML3603.0;
(* Rung L57 *)
%QX1.4.23 := NOT (NOT %QX2.3.0 AND NOT %QX2.3.4 AND NOT %IX2.0.1 AND NOT %IX2.0.9) AND NOT %ML3603.0;
(* Rung L58 *)
%QX1.4.24 := NOT (NOT %QX3.3.0 AND NOT %QX3.3.4 AND NOT %IX3.0.1 AND NOT %IX3.0.9) AND NOT %ML3603.0;

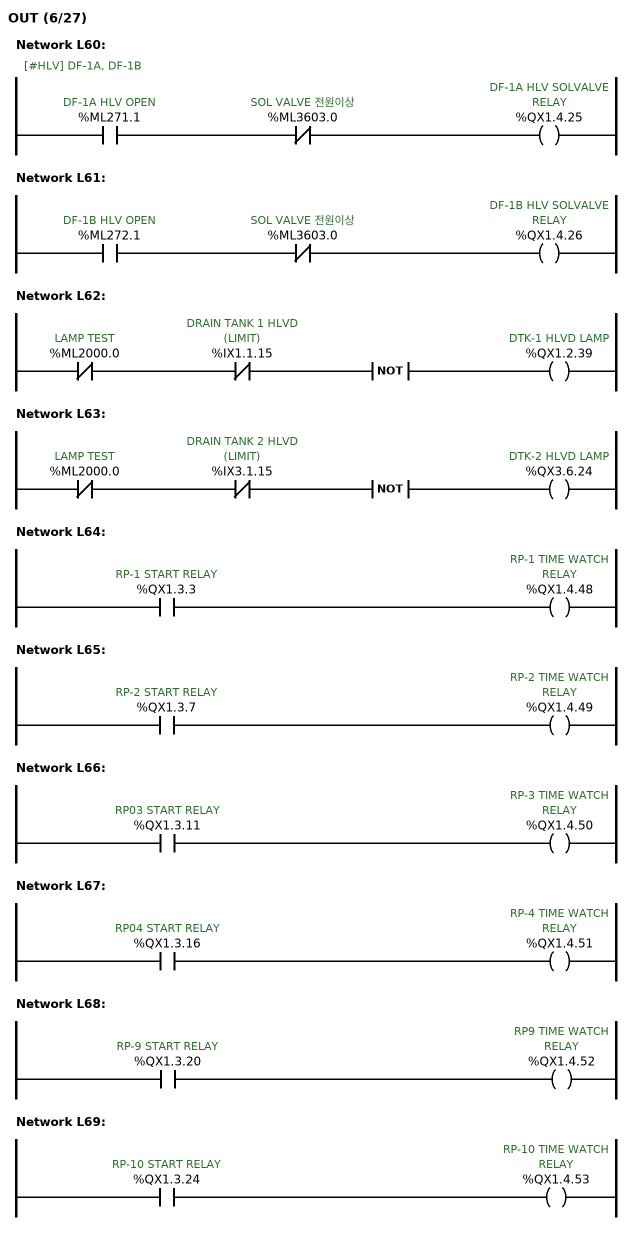
(* [#HLV] DF-1A, DF-1B *)
(* Rung L60 *)
%QX1.4.25 := %ML271.1 AND NOT %ML3603.0;
(* Rung L61 *)
%QX1.4.26 := %ML272.1 AND NOT %ML3603.0;
(* Rung L62 *)
%QX1.2.39 := NOT (NOT %ML2000.0 AND NOT %IX1.1.15);
(* Rung L63 *)
%QX3.6.24 := NOT (NOT %ML2000.0 AND NOT %IX3.1.15);
(* Rung L64 *)
%QX1.4.48 := %QX1.3.3;
(* Rung L65 *)
%QX1.4.49 := %QX1.3.7;
(* Rung L66 *)
%QX1.4.50 := %QX1.3.11;
(* Rung L67 *)
%QX1.4.51 := %QX1.3.16;
(* Rung L68 *)
%QX1.4.52 := %QX1.3.20;
(* Rung L69 *)
%QX1.4.53 := %QX1.3.24;

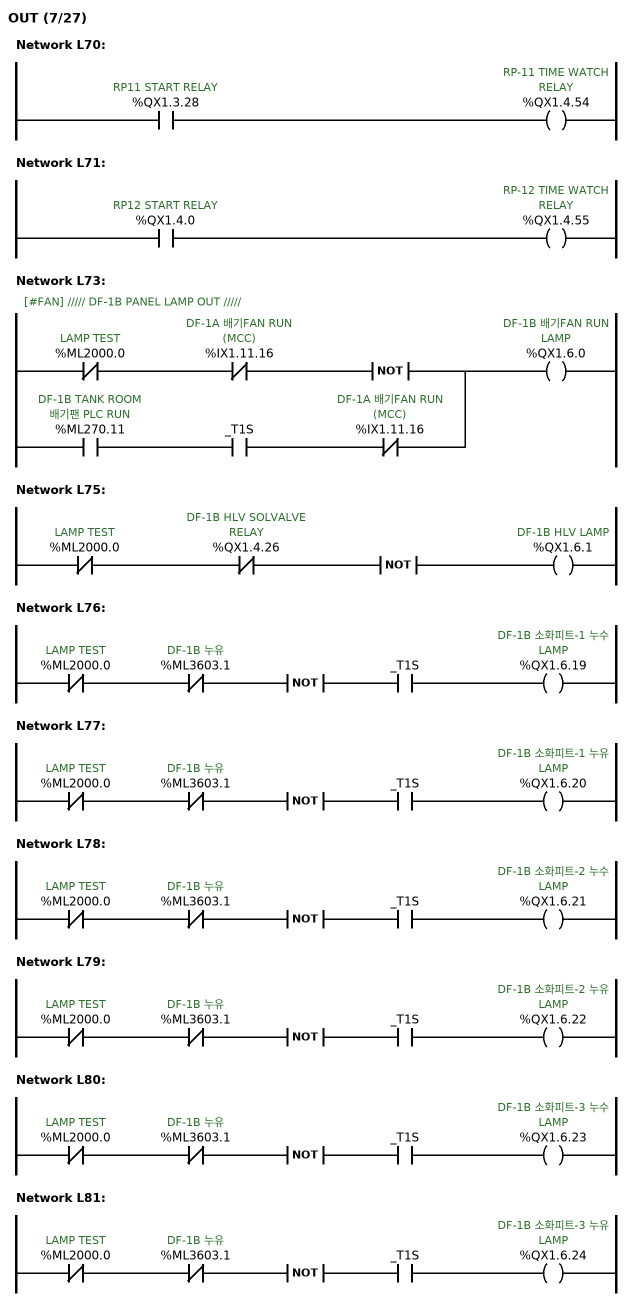
(* Rung L70 *)
%QX1.4.54 := %QX1.3.28;
(* Rung L71 *)
%QX1.4.55 := %QX1.4.0;
(* [#FAN] ///// DF-1B PANEL LAMP OUT ///// *)
(* Rung L73 *)
%QX1.6.0 := NOT (NOT %ML2000.0 AND NOT %IX1.11.16) OR (%ML270.11 AND _T1S AND NOT %IX1.11.16);
(* Rung L75 *)
%QX1.6.1 := NOT (NOT %ML2000.0 AND NOT %QX1.4.26);
(* Rung L76 *)
%QX1.6.19 := NOT (NOT %ML2000.0 AND NOT %ML3603.1) AND _T1S;
(* Rung L77 *)
%QX1.6.20 := NOT (NOT %ML2000.0 AND NOT %ML3603.1) AND _T1S;
(* Rung L78 *)
%QX1.6.21 := NOT (NOT %ML2000.0 AND NOT %ML3603.1) AND _T1S;
(* Rung L79 *)
%QX1.6.22 := NOT (NOT %ML2000.0 AND NOT %ML3603.1) AND _T1S;
(* Rung L80 *)
%QX1.6.23 := NOT (NOT %ML2000.0 AND NOT %ML3603.1) AND _T1S;
(* Rung L81 *)
%QX1.6.24 := NOT (NOT %ML2000.0 AND NOT %ML3603.1) AND _T1S;

